FUNCTION_BLOCK FB_VirtualControlBox IMPLEMENTS I_ControlBox
VAR_INPUT
END_VAR
VAR_OUTPUT
END_VAR
VAR
END_VAR

METHOD Lamps
VAR_INPUT
	bEnable : BOOL;
END_VAR
IF bEnable THEN 
	G_VirtualControlBox.bGreenLight := G_Work.bRunning;
	G_VirtualControlBox.bRedLight := G_Work.bFault;
END_IF
END_METHOD

METHOD ModeSelector 
VAR_INPUT
END_VAR
VAR_OUTPUT
	eMode : E_Mode;
END_VAR
CASE eMode OF 
	E_Mode.Off:	
		IF G_VirtualControlBox.bOnSelector AND NOT(G_VirtualControlBox.bAutoSelector) THEN	
			eMode := E_Mode.Manual;
		END_IF
		
		IF G_VirtualControlBox.bOnSelector AND G_VirtualControlBox.bAutoSelector THEN	
			eMode := E_Mode.Auto;
		END_IF

	E_Mode.Manual: 
		IF NOT(G_VirtualControlBox.bOnSelector) THEN	
			eMode := E_Mode.Off;
		END_IF
		
		IF G_VirtualControlBox.bOnSelector AND G_VirtualControlBox.bAutoSelector THEN	
			eMode := E_Mode.Auto;
		END_IF
	
	E_Mode.Auto:
		IF NOT(G_VirtualControlBox.bOnSelector) THEN	
			eMode := E_Mode.Off;
		END_IF
		
		IF G_VirtualControlBox.bOnSelector AND NOT(G_VirtualControlBox.bAutoSelector) THEN	
			eMode := E_Mode.Manual;
		END_IF	
ELSE 	
	eMode := E_Mode.Off;
END_CASE
END_METHOD

END_FUNCTION_BLOCK

(* stored: Version 1.1.0.1, ProductVersion 3.1.4024.10
   POU FB_VirtualControlBox: Id {b5dbd877-8357-49f5-a98a-ac539e1b1d21}, SpecialFunc None
   Method Lamps: Id {0dd9b505-9eff-424c-bfde-77014d6169c5}
   Method ModeSelector: Id {e15f3617-ec38-4567-aa4b-7e33c463052d} *)
